// TIA Portal V20 export
DATA_BLOCK "Instance_FB_Frequency_Inverter_DB_Spin_Caroussel"   // DB106
// stored: AutoNumber false, InstanceOfName FB_Frequency_Inverter, InstanceOfType FB
"FB_Frequency_Inverter"
   // VAR_INPUT
   //    Emergency_Stop_Release : Bool;
   //    Start : Bool;
   //    Manual_Turn_On_Motor : Bool;
   //    Pause_Conveyor_Belt_And_Carousel_Functional_Test : Bool;
   //    Select_Motor_Speedy : SInt;
   // END_VAR
   // VAR_OUTPUT
   //    Motor_Spining_Speedy_1 : Bool;
   //    Motor_Spining_Speedy_2 : Bool;
   //    Motor_Spining_Speedy_3 : Bool;
   // END_VAR
BEGIN
END_DATA_BLOCK
